// TwinCAT 3 PLC project ReferenceImplementation
// ProgramVersion: 3.1.4026.11
// libraries:
//   Tc2_Standard, * (Beckhoff Automation GmbH)
//   Tc2_System, * (Beckhoff Automation GmbH)
//   Tc3_Module, * (Beckhoff Automation GmbH)
//   [Resi4MPM], * (Jan Wilch)
//   [xPPU], * (Jan Wilch)
// project tree:
//   DUTs/ SRecoveryRequestOutput.TcDUT, STriggeredOutput.TcDUT
//   GVLs/ HMI_Texts.TcGVL, RaInterface_GVL.TcGVL (excluded from build), xPPU_Container.TcPOU
//   / PlcTask.TcTTO
//   POUs/00_ProgramMain/ MAIN.TcPOU
//   POUs/01_SequenceControl/ xPPU_Automatic.TcPOU, xPPU_LSC.TcPOU, xPPU_Crane.TcPOU, xPPU_PAC.TcPOU, xPPU_PicAlpha.TcPOU, xPPU_RFC.TcPOU, xPPU_SSC.TcPOU, xPPU_Stack.TcPOU, xPPU_Stamp.TcPOU
//   POUs/98_Utility/ FC_InitAlarmTexts.TcPOU
//   POUs/99_ExtrafunctionalImpl/ ButtonManager.TcPOU
// real-time tasks:
//   TASK PlcTask: cycle T#10ms, priority 20, ADS port 351
// I/O:
//   DEVICE Device 1 (EtherCAT), AmsNetId 192.168.5.90.2.1
//     Term 84 (EK1200) [EK1200-5000 EtherCAT Power supply (2A E-Bus)]
//       Term 2 (EK1110) [EK1110 EtherCAT extension]
//     BK1 (EK1100) [EK1100 EtherCAT Coupler (2A E-Bus)]
//       1.2 (EL1004) [EL1004 4Ch. Dig. Input 24V, 3ms]
//       1.3 (EL1004) [EL1004 4Ch. Dig. Input 24V, 3ms]
//       1.4 (EL1004) [EL1004 4Ch. Dig. Input 24V, 3ms]
//       1.5 (EL1004) [EL1004 4Ch. Dig. Input 24V, 3ms]
//       1.6 (EL2004) [EL2004 4Ch. Dig. Output 24V, 0.5A]
//       1.9 (EL2004) [EL2004 4Ch. Dig. Output 24V, 0.5A]
//       1.10 (EL2004) [EL2004 4Ch. Dig. Output 24V, 0.5A]
//       1.11 (EL2004) [EL2004 4Ch. Dig. Output 24V, 0.5A]
//       1.12 (EL1004) [EL1004 4Ch. Dig. Input 24V, 3ms]
//       1.13 (EL3162) [EL3162 2Ch. Ana. Input 0-10V]
//       1.14 (EL9011) [EL9011 End Terminal]
//     BK2&3 (EK1100) [EK1100 EtherCAT Coupler (2A E-Bus)]
//       2&3.2 (EL1004) [EL1004 4Ch. Dig. Input 24V, 3ms]
//       2&3.3 (EL1004) [EL1004 4Ch. Dig. Input 24V, 3ms]
//       2&3.4 (EL1004) [EL1004 4Ch. Dig. Input 24V, 3ms]
//       2&3.5 (EL1004) [EL1004 4Ch. Dig. Input 24V, 3ms]
//       2&3.6 (EL1004) [EL1004 4Ch. Dig. Input 24V, 3ms]
//       2&3.7 (EL1004) [EL1004 4Ch. Dig. Input 24V, 3ms]
//       2&3.10 (EL2004) [EL2004 4Ch. Dig. Output 24V, 0.5A]
//       2&3.11 (EL2004) [EL2004 4Ch. Dig. Output 24V, 0.5A]
//       2&3.12 (EL2004) [EL2004 4Ch. Dig. Output 24V, 0.5A]
//       2&3.13 (EL2004) [EL2004 4Ch. Dig. Output 24V, 0.5A]
//       2&3.14 (EL1004) [EL1004 4Ch. Dig. Input 24V, 3ms]
//       2&3.16 (EL4102) [EL4102 2Ch. Ana. Output 0-10V]
//       2&3.17 (EL4102) [EL4102 2Ch. Ana. Output 0-10V]
//       2&3.18 (EL9011) [EL9011 End Terminal]
//     BK4 (EK1100) [EK1100 EtherCAT Coupler (2A E-Bus)]
//       4.2 (EL1808) [EL1808 8Ch. Dig. Input 24V, 3ms]
//       4.3 (EL1004) [EL1004 4Ch. Dig. Input 24V, 3ms]
//       4.4 (EL1004) [EL1004 4Ch. Dig. Input 24V, 3ms]
//       4.5 (EL1004) [EL1004 4Ch. Dig. Input 24V, 3ms]
//       4.6 (EL1004) [EL1004 4Ch. Dig. Input 24V, 3ms]
//       4.7 (EL1004) [EL1004 4Ch. Dig. Input 24V, 3ms]
//       4.8 (EL3064) [EL3064 4Ch. Ana. Input 0-10V]
//       4.9 (EL3064) [EL3064 4Ch. Ana. Input 0-10V]
//       4.10 (EL3164) [EL3164 4Ch. Ana. Input 0-10V]
//       4.11 (EL3054) [EL3054 4Ch. Ana. Input 4-20mA]
//       Term 208 (EL3058) [EL3058 8Ch. Ana. Input 4-20mA]
//       4.13 (EL2004) [EL2004 4Ch. Dig. Output 24V, 0.5A]
//       4.14 (EL2004) [EL2004 4Ch. Dig. Output 24V, 0.5A]
//       4.15 (EL9011) [EL9011 End Terminal]
//     BK5 (EK1100) [EK1100 EtherCAT Coupler (2A E-Bus)]
//       5.2 (EL1008) [EL1008 8Ch. Dig. Input 24V, 3ms]
//       5.3 (EL5152) [EL5152 2Ch. Inc. Encoder]
//       5.6 (EL2008) [EL2008 8Ch. Dig. Output 24V, 0.5A]
//       5.7 (EL4102) [EL4102 2Ch. Ana. Output 0-10V]
//       5.8 (EL9011) [EL9011 End Terminal]
//     BK6 (EK1100) [EK1100 EtherCAT Coupler (2A E-Bus)]
//       6.2 (EL3062) [EL3062 2Ch. Ana. Input 0-10V]
//       6.3 (EL6224) [EL6224 (IO Link Master)]
//       6.4 (EL9011) [EL9011 End Terminal]
//     BK7 (EK1100) [EK1100 EtherCAT Coupler (2A E-Bus)]
//       7.2 (EL1004) [EL1004 4Ch. Dig. Input 24V, 3ms]
//       7.5 (EL2004) [EL2004 4Ch. Dig. Output 24V, 0.5A]
//       7.8 (EL6224) [EL6224 (IO Link Master)]
//       7.9 (EL9011) [EL9011 End Terminal]
//     BK8 (EK1100) [EK1100 EtherCAT Coupler (2A E-Bus)]
//       8.2 (EL1008) [EL1008 8Ch. Dig. Input 24V, 3ms]
//       8.3 (EL1004) [EL1004 4Ch. Dig. Input 24V, 3ms]
//       8.4 (EL3062) [EL3062 2Ch. Ana. Input 0-10V]
//       8.5 (EL2004) [EL2004 4Ch. Dig. Output 24V, 0.5A]
//       8.8 (EL2008) [EL2008 8Ch. Dig. Output 24V, 0.5A]
//       8.9 (EL2004) [EL2004 4Ch. Dig. Output 24V, 0.5A]
//       Term 114 (EL1808) [EL1808 8Ch. Dig. Input 24V, 3ms]
//       8.10 (EL9011) [EL9011 End Terminal]
//     BK9 (EK1100) [EK1100 EtherCAT Coupler (2A E-Bus)]
//       9.2 (EL1004) [EL1004 4Ch. Dig. Input 24V, 3ms]
//       9.3 (EL5152) [EL5152 2Ch. Inc. Encoder]
//       9.6 (EL2004) [EL2004 4Ch. Dig. Output 24V, 0.5A]
//       9.7 (EL4102) [EL4102 2Ch. Ana. Output 0-10V]
//       9.8 (EL9011) [EL9011 End Terminal]
//     BK10 (EK1100) [EK1100 EtherCAT Coupler (2A E-Bus)]
//       10.2 (EL1004) [EL1004 4Ch. Dig. Input 24V, 3ms]
//       10.3 (EL5152) [EL5152 2Ch. Inc. Encoder]
//       10.6 (EL2004) [EL2004 4Ch. Dig. Output 24V, 0.5A]
//       10.7 (EL4102) [EL4102 2Ch. Ana. Output 0-10V]
//       10.8 (EL9011) [EL9011 End Terminal]
//     BK11 (EK1100) [EK1100 EtherCAT Coupler (2A E-Bus)]
//       11.2 (EL1004) [EL1004 4Ch. Dig. Input 24V, 3ms]
//       11.3 (EL3064) [EL3064 4Ch. Ana. Input 0-10V]
//       11.6 (EL2004) [EL2004 4Ch. Dig. Output 24V, 0.5A]
//       11.7 (EL9011) [EL9011 End Terminal]
// variable links:
//   ReferenceImplementation/ReferenceImplementation Instance <-> Device 1 (EtherCAT)/BK1 (EK1100)/1.10 (EL2004)
//     PlcTask Outputs/MAIN.m_container.m_crane.Motor.DO_TurnClockwise <-> Channel 4/Output
//     PlcTask Outputs/MAIN.m_container.m_crane.Motor.DO_TurnCounterclockwise <-> Channel 3/Output
//   ReferenceImplementation/ReferenceImplementation Instance <-> Device 1 (EtherCAT)/BK1 (EK1100)/1.2 (EL1004)
//     PlcTask Inputs/MAIN.m_buttonManager.DI_AutomaticSwitch_StackTerminal <-> Channel 3/Input
//     PlcTask Inputs/MAIN.m_buttonManager.DI_EStopButton_Terminal1 <-> Channel 1/Input
//     PlcTask Inputs/MAIN.m_buttonManager.DI_StartButton_Terminal1 <-> Channel 2/Input
//     PlcTask Inputs/MAIN.m_container.m_crane.o_VacuumGripper.DI_TakenIn <-> Channel 4/Input
//   ReferenceImplementation/ReferenceImplementation Instance <-> Device 1 (EtherCAT)/BK1 (EK1100)/1.3 (EL1004)
//     PlcTask Inputs/MAIN.m_container.m_crane.o_MonostableCylinder.DI_Extended <-> Channel 1/Input
//     PlcTask Inputs/MAIN.m_container.m_crane.o_MonostableCylinder.DI_Retracted <-> Channel 2/Input
//     PlcTask Inputs/MAIN.m_container.m_stack.o_slidingCylinder.DI_Extended <-> Channel 4/Input
//     PlcTask Inputs/MAIN.m_container.m_stack.o_slidingCylinder.DI_Retracted <-> Channel 3/Input
//   ReferenceImplementation/ReferenceImplementation Instance <-> Device 1 (EtherCAT)/BK1 (EK1100)/1.4 (EL1004)
//     PlcTask Inputs/MAIN.m_container.m_crane.m_PresenceSensorAtConveyor.DI_WPDetected <-> Channel 4/Input
//     PlcTask Inputs/MAIN.m_container.m_crane.m_PresenceSensorAtStamp.DI_WPDetected <-> Channel 3/Input
//     PlcTask Inputs/MAIN.m_container.m_stack.m_Inductivesensor.DI_WPMetallic <-> Channel 1/Input
//     PlcTask Inputs/MAIN.m_container.m_stack.m_Opticalsensor.DI_WPLight <-> Channel 2/Input
//   ReferenceImplementation/ReferenceImplementation Instance <-> Device 1 (EtherCAT)/BK1 (EK1100)/1.5 (EL1004)
//     PlcTask Inputs/MAIN.m_container.m_crane.m_PresenceSensorAtStack.DI_WPDetected <-> Channel 1/Input
//     PlcTask Inputs/MAIN.m_container.m_stack.m_Presencesensor.DI_WPDetected <-> Channel 2/Input
//   ReferenceImplementation/ReferenceImplementation Instance <-> Device 1 (EtherCAT)/BK1 (EK1100)/1.6 (EL2004)
//     PlcTask Outputs/MAIN.m_container.m_crane.o_VacuumGripper.DO_VacuumOn <-> Channel 1/Output
//   ReferenceImplementation/ReferenceImplementation Instance <-> Device 1 (EtherCAT)/BK1 (EK1100)/1.9 (EL2004)
//     PlcTask Outputs/MAIN.m_container.m_crane.o_MonostableCylinder.DO_Extend <-> Channel 1/Output
//     PlcTask Outputs/MAIN.m_container.m_stack.o_slidingCylinder.DO_Extend <-> Channel 2/Output
//   ReferenceImplementation/ReferenceImplementation Instance <-> Device 1 (EtherCAT)/BK10 (EK1100)/10.2 (EL1004)
//     PlcTask Inputs/MAIN.m_container.m_SSC.m_PresencesensorEnd.DI_WPDetected <-> Channel 2/Input
//     PlcTask Inputs/MAIN.m_container.m_SSC.m_PresencesensorStart.DI_WPDetected <-> Channel 1/Input
//     PlcTask Inputs/MAIN.m_container.m_SSC.m_Switch.DI_Extended <-> Channel 4/Input
//     PlcTask Inputs/MAIN.m_container.m_SSC.m_Switch.DI_Retracted <-> Channel 3/Input
//   ReferenceImplementation/ReferenceImplementation Instance <-> Device 1 (EtherCAT)/BK10 (EK1100)/10.6 (EL2004)
//     PlcTask Outputs/MAIN.m_container.m_SSC.Motor.DO_TurnClockwise <-> Channel 1/Output
//     PlcTask Outputs/MAIN.m_container.m_SSC.Motor.DO_TurnCounterclockwise <-> Channel 2/Output
//     PlcTask Outputs/MAIN.m_container.m_SSC.m_Switch.DO_Extend <-> Channel 3/Output
//   ReferenceImplementation/ReferenceImplementation Instance <-> Device 1 (EtherCAT)/BK2&3 (EK1100)/2&3.10 (EL2004)
//     PlcTask Outputs/MAIN.m_container.m_stamp.m_slidingCylinder.DO_Extend <-> Channel 1/Output
//     PlcTask Outputs/MAIN.m_container.m_stamp.m_slidingCylinder.DO_Retract <-> Channel 2/Output
//     PlcTask Outputs/MAIN.m_container.m_stamp.m_stampingCylinder.DO_Extend <-> Channel 3/Output
//   ReferenceImplementation/ReferenceImplementation Instance <-> Device 1 (EtherCAT)/BK2&3 (EK1100)/2&3.11 (EL2004)
//     PlcTask Outputs/MAIN.m_container.m_LSC.Motor.DO_TurnClockwise <-> Channel 4/Output
//     PlcTask Outputs/MAIN.m_container.m_LSC.m_rampPusherMid.DO_Extend <-> Channel 3/Output
//     PlcTask Outputs/MAIN.m_container.m_LSC.m_rampPusherStart.DO_Extend <-> Channel 2/Output
//   ReferenceImplementation/ReferenceImplementation Instance <-> Device 1 (EtherCAT)/BK2&3 (EK1100)/2&3.12 (EL2004)
//     PlcTask Outputs/MAIN.m_container.m_LSC.Motor.DO_TurnCounterclockwise <-> Channel 1/Output
//   ReferenceImplementation/ReferenceImplementation Instance <-> Device 1 (EtherCAT)/BK2&3 (EK1100)/2&3.16 (EL4102)
//     PlcTask Outputs/MAIN.m_container.m_stamp.m_pressureValve.AO_SetPressure <-> Channel 2/Output
//   ReferenceImplementation/ReferenceImplementation Instance <-> Device 1 (EtherCAT)/BK2&3 (EK1100)/2&3.2 (EL1004)
//     PlcTask Inputs/MAIN.m_buttonManager.DI_AutomaticSwitch_StampTerminal <-> Channel 1/Input
//     PlcTask Inputs/MAIN.m_container.m_stamp.m_slidingCylinder.DI_Extended <-> Channel 2/Input
//     PlcTask Inputs/MAIN.m_container.m_stamp.m_slidingCylinder.DI_Retracted <-> Channel 3/Input
//     PlcTask Inputs/MAIN.m_container.m_stamp.m_stampingCylinder.DI_Retracted <-> Channel 4/Input
//   ReferenceImplementation/ReferenceImplementation Instance <-> Device 1 (EtherCAT)/BK2&3 (EK1100)/2&3.3 (EL1004)
//     PlcTask Inputs/MAIN.m_buttonManager.DI_EStopButton_Terminal3 <-> Channel 3/Input
//     PlcTask Inputs/MAIN.m_buttonManager.DI_StartButton_Terminal3 <-> Channel 4/Input
//     PlcTask Inputs/MAIN.m_container.m_stamp.m_presenceSensor.DI_WPDetected <-> Channel 2/Input
//     PlcTask Inputs/MAIN.m_container.m_stamp.m_stampingCylinder.DI_Extended <-> Channel 1/Input
//   ReferenceImplementation/ReferenceImplementation Instance <-> Device 1 (EtherCAT)/BK2&3 (EK1100)/2&3.4 (EL1004)
//     PlcTask Inputs/MAIN.m_buttonManager.DI_AutomaticSwitch_LSCTerminal <-> Channel 1/Input
//     PlcTask Inputs/MAIN.m_container.m_LSC.m_inductiveSensorStart.DI_WPMetallic <-> Channel 4/Input
//     PlcTask Inputs/MAIN.m_container.m_LSC.m_presenceSensorStart.DI_WPDetected <-> Channel 3/Input
//   ReferenceImplementation/ReferenceImplementation Instance <-> Device 1 (EtherCAT)/BK2&3 (EK1100)/2&3.5 (EL1004)
//     PlcTask Inputs/MAIN.m_container.m_LSC.m_inductiveSensorMid.DI_WPMetallic <-> Channel 2/Input
//     PlcTask Inputs/MAIN.m_container.m_LSC.m_opticalSensorEnd.DI_WPLight <-> Channel 4/Input
//     PlcTask Inputs/MAIN.m_container.m_LSC.m_opticalSensorMid.DI_WPLight <-> Channel 3/Input
//     PlcTask Inputs/MAIN.m_container.m_LSC.m_opticalSensorStart.DI_WPLight <-> Channel 1/Input
//   ReferenceImplementation/ReferenceImplementation Instance <-> Device 1 (EtherCAT)/BK2&3 (EK1100)/2&3.6 (EL1004)
//     PlcTask Inputs/MAIN.m_container.m_LSC.m_rampPusherMid.DI_Extended <-> Channel 3/Input
//     PlcTask Inputs/MAIN.m_container.m_LSC.m_rampPusherMid.DI_Retracted <-> Channel 4/Input
//     PlcTask Inputs/MAIN.m_container.m_LSC.m_rampPusherStart.DI_Extended <-> Channel 1/Input
//     PlcTask Inputs/MAIN.m_container.m_LSC.m_rampPusherStart.DI_Retracted <-> Channel 2/Input
//   ReferenceImplementation/ReferenceImplementation Instance <-> Device 1 (EtherCAT)/BK2&3 (EK1100)/2&3.7 (EL1004)
//     PlcTask Inputs/MAIN.m_buttonManager.DI_EStopButton_Terminal2 <-> Channel 3/Input
//     PlcTask Inputs/MAIN.m_buttonManager.DI_StartButton_Terminal2 <-> Channel 4/Input
//   ReferenceImplementation/ReferenceImplementation Instance <-> Device 1 (EtherCAT)/BK4 (EK1100)/4.2 (EL1808)
//     PlcTask Inputs/MAIN.m_container.m_LSC.m_rampEnd.m_presenceSensorRampFull.DI_WPDetected <-> Channel 8/Input
//     PlcTask Inputs/MAIN.m_container.m_LSC.m_rampMiddle.m_presenceSensorRampFull.DI_WPDetected <-> Channel 7/Input
//     PlcTask Inputs/MAIN.m_container.m_LSC.m_rampStart.m_presenceSensorRampFull.DI_WPDetected <-> Channel 6/Input
//   ReferenceImplementation/ReferenceImplementation Instance <-> Device 1 (EtherCAT)/BK4 (EK1100)/4.3 (EL1004)
//     PlcTask Inputs/MAIN.m_container.m_stack.o_slidingCylinder.DI_BoundaryPressure <-> Channel 1/Input
//     PlcTask Inputs/MAIN.m_container.m_stamp.m_slidingCylinder.DI_BoundaryPressure <-> Channel 2/Input
//   ReferenceImplementation/ReferenceImplementation Instance <-> Device 1 (EtherCAT)/BK4 (EK1100)/4.4 (EL1004)
//     PlcTask Inputs/MAIN.m_container.m_stamp.m_stampingCylinder.DI_BoundaryPressure <-> Channel 4/Input
//   ReferenceImplementation/ReferenceImplementation Instance <-> Device 1 (EtherCAT)/BK4 (EK1100)/4.5 (EL1004)
//     PlcTask Inputs/MAIN.m_container.m_SSC.m_Inductivesensor.DI_WPMetallic <-> Channel 2/Input
//     PlcTask Inputs/MAIN.m_container.m_SSC.m_Opticalsensor.DI_WPLight <-> Channel 1/Input
//     PlcTask Inputs/MAIN.m_container.m_SSC.m_Ramp.m_presenceSensorRampFull.DI_WPDetected <-> Channel 3/Input
//   ReferenceImplementation/ReferenceImplementation Instance <-> Device 1 (EtherCAT)/BK4 (EK1100)/4.6 (EL1004)
//     PlcTask Inputs/MAIN.m_container.m_stamp.m_stampingCylinder.DI_BoundaryFlowPressure <-> Channel 1/Input
//   ReferenceImplementation/ReferenceImplementation Instance <-> Device 1 (EtherCAT)/BK4 (EK1100)/4.9 (EL3064)
//     PlcTask Inputs/MAIN.m_container.m_stamp.m_pressureSensor.AI_CurrentPressure <-> AI Standard Channel 2/Value
//   ReferenceImplementation/ReferenceImplementation Instance <-> Device 1 (EtherCAT)/BK5 (EK1100)/5.2 (EL1008)
//     PlcTask Inputs/MAIN.m_buttonManager.DI_AutomaticSwitch_DoorTerminal <-> Channel 3/Input
//     PlcTask Inputs/MAIN.m_buttonManager.DI_ResetButton_Door <-> Channel 4/Input
//     PlcTask Inputs/MAIN.m_buttonManager.DI_StartButton_Door <-> Channel 1/Input
//     PlcTask Inputs/MAIN.m_buttonManager.DI_StopButton_Door <-> Channel 2/Input
//     PlcTask Inputs/MAIN.m_container.m_RFC.m_PresencesensorEnd.DI_WPDetected <-> Channel 6/Input
//     PlcTask Inputs/MAIN.m_container.m_RFC.m_PresencesensorStart.DI_WPDetected <-> Channel 5/Input
//     PlcTask Inputs/MAIN.m_container.m_RFC.m_Switch.DI_Extended <-> Channel 8/Input
//     PlcTask Inputs/MAIN.m_container.m_RFC.m_Switch.DI_Retracted <-> Channel 7/Input
//   ReferenceImplementation/ReferenceImplementation Instance <-> Device 1 (EtherCAT)/BK5 (EK1100)/5.6 (EL2008)
//     PlcTask Outputs/MAIN.m_container.m_RFC.Motor.DO_TurnClockwise <-> Channel 5/Output
//     PlcTask Outputs/MAIN.m_container.m_RFC.Motor.DO_TurnCounterclockwise <-> Channel 6/Output
//     PlcTask Outputs/MAIN.m_container.m_RFC.m_Switch.DO_Extend <-> Channel 7/Output
//   ReferenceImplementation/ReferenceImplementation Instance <-> Device 1 (EtherCAT)/BK6 (EK1100)/6.2 (EL3062)
//     PlcTask Inputs/MAIN.m_container.m_stack.m_Weightsensor.AI_WPWeight <-> AI Standard Channel 1/Value
//   ReferenceImplementation/ReferenceImplementation Instance <-> Device 1 (EtherCAT)/BK7 (EK1100)/7.5 (EL2004)
//     PlcTask Outputs/MAIN.m_container.m_LSC.m_Switch.DO_Extend <-> Channel 3/Output
//   ReferenceImplementation/ReferenceImplementation Instance <-> Device 1 (EtherCAT)/BK8 (EK1100)/8.2 (EL1008)
//     PlcTask Inputs/MAIN.m_buttonManager.DI_EStopButton_LightBarrier <-> Channel 8/Input
//     PlcTask Inputs/MAIN.m_container.m_PicAlpha.m_PresenceSensorPosition1.DI_WPDetected <-> Channel 2/Input
//     PlcTask Inputs/MAIN.m_container.m_PicAlpha.m_PresenceSensorPosition2.DI_WPDetected <-> Channel 7/Input
//     PlcTask Inputs/MAIN.m_container.m_PicAlpha.m_PresenceSensorPosition3.DI_WPDetected <-> Channel 4/Input
//     PlcTask Inputs/MAIN.m_container.m_PicAlpha.m_PresenceSensorPosition4.DI_WPDetected <-> Channel 3/Input
//     PlcTask Inputs/MAIN.m_container.m_PicAlpha.o_MonostableCylinder.DI_Extended <-> Channel 5/Input
//     PlcTask Inputs/MAIN.m_container.m_PicAlpha.o_MonostableCylinder.DI_Retracted <-> Channel 6/Input
//     PlcTask Inputs/MAIN.m_container.m_PicAlpha.o_VacuumGripper.DI_TakenIn <-> Channel 1/Input
//   ReferenceImplementation/ReferenceImplementation Instance <-> Device 1 (EtherCAT)/BK8 (EK1100)/8.3 (EL1004)
//     PlcTask Inputs/MAIN.m_buttonManager.DI_AutomaticSwitch_LightGridTerminal <-> Channel 3/Input
//     PlcTask Inputs/MAIN.m_buttonManager.DI_ResetButton_LightBarrier <-> Channel 4/Input
//     PlcTask Inputs/MAIN.m_buttonManager.DI_StartButton_LightBarrier <-> Channel 1/Input
//     PlcTask Inputs/MAIN.m_buttonManager.DI_StopButton_LightBarrier <-> Channel 2/Input
//   ReferenceImplementation/ReferenceImplementation Instance <-> Device 1 (EtherCAT)/BK8 (EK1100)/8.5 (EL2004)
//     PlcTask Outputs/MAIN.m_container.m_PicAlpha.o_VacuumGripper.DO_VacuumOn <-> Channel 1/Output
//   ReferenceImplementation/ReferenceImplementation Instance <-> Device 1 (EtherCAT)/BK8 (EK1100)/8.8 (EL2008)
//     PlcTask Outputs/MAIN.m_container.m_PicAlpha.Motor.DO_TurnClockwise <-> Channel 2/Output
//     PlcTask Outputs/MAIN.m_container.m_PicAlpha.Motor.DO_TurnCounterclockwise <-> Channel 1/Output
//     PlcTask Outputs/MAIN.m_container.m_PicAlpha.o_MonostableCylinder.DO_Extend <-> Channel 3/Output
//     PlcTask Outputs/MAIN.m_container.m_PicAlpha.o_VacuumGripper.VacuumHit <-> Channel 6/Output
//   ReferenceImplementation/ReferenceImplementation Instance <-> Device 1 (EtherCAT)/BK9 (EK1100)/9.2 (EL1004)
//     PlcTask Inputs/MAIN.m_container.m_PAC.m_PresencesensorEnd.DI_WPDetected <-> Channel 2/Input
//     PlcTask Inputs/MAIN.m_container.m_PAC.m_PresencesensorStart.DI_WPDetected <-> Channel 1/Input
//     PlcTask Inputs/MAIN.m_container.m_PAC.m_Switch.DI_Extended <-> Channel 4/Input
//     PlcTask Inputs/MAIN.m_container.m_PAC.m_Switch.DI_Retracted <-> Channel 3/Input
//   ReferenceImplementation/ReferenceImplementation Instance <-> Device 1 (EtherCAT)/BK9 (EK1100)/9.6 (EL2004)
//     PlcTask Outputs/MAIN.m_container.m_PAC.Motor.DO_TurnClockwise <-> Channel 1/Output
//     PlcTask Outputs/MAIN.m_container.m_PAC.Motor.DO_TurnCounterclockwise <-> Channel 2/Output
//     PlcTask Outputs/MAIN.m_container.m_PAC.m_Switch.DO_Extend <-> Channel 3/Output

CONFIGURATION ReferenceImplementation
    RESOURCE PLC ON TwinCAT3
        TASK PlcTask(INTERVAL := T#10ms, PRIORITY := 20);
        PROGRAM MAIN WITH PlcTask : MAIN;
    END_RESOURCE
END_CONFIGURATION

// ---- DUTs/SRecoveryRequestOutput.TcDUT
TYPE SRecoveryRequestOutput EXTENDS STriggeredOutput :
STRUCT
	RequestedState: STRING(256);
END_STRUCT
END_TYPE

// ---- DUTs/STriggeredOutput.TcDUT
TYPE STriggeredOutput :
STRUCT
	ChangeTrigger: USINT;
END_STRUCT
END_TYPE

// ---- GVLs/HMI_Texts.TcGVL
{attribute 'qualified_only'}
VAR_GLOBAL
	AlarmTexts: ARRAY [0..999] OF STRING;
END_VAR

// ---- GVLs/RaInterface_GVL.TcGVL
{attribute 'qualified_only'}
VAR_GLOBAL CONSTANT
	ALARM_ARR_MAX: UINT := 9;
END_VAR

VAR_GLOBAL
	// #################### OUTPUT TO RA ####################
	// alarms detected at field-level or process-level (irregularly pushed to RA)
	{attribute 'OPC.UA.DA' := '1'}
	Out_Alarms: ARRAY [ResiConst.ARR_MIN..RaInterface_GVL.ALARM_ARR_MAX] OF SAlarm;
	
	// the complete set of observed process variables (explicitly checked by RA)
	{attribute 'OPC.UA.DA' := '1'}
	Out_NamedProcessState: ARRAY [ResiConst.ARR_MIN..ResiConst.STATE_ARR_MAX] OF SNamedValue;
	
	// the process state that needs to be restored (irregularly pushed to RA)
	{attribute 'OPC.UA.DA' := '1'}
	{attribute 'OPC.UA.DA.StructuredType' := '1'}
	Out_RecoveryRequest: SRecoveryRequestOutput;
	
	
	// ################### INPUT FROM RA ####################
	// CPA-computed specifications of compensation strategies
	{attribute 'OPC.UA.DA' := '1'}
	In_Compensations: ARRAY [ResiConst.ARR_MIN..ResiConst.COMPENSATIONS_ARR_MAX] OF SCompensation;
	
	// CPA-computed specification of a recovery strategy
	{attribute 'OPC.UA.DA' := '1'}
	{attribute 'OPC.UA.DA.StructuredType' := '1'}
	In_Recovery: SRecovery;
	
	// specifies whether a recovery is ready for execution
	{attribute 'OPC.UA.DA' := '1'}
	In_RecoveryAvailable: BOOL;
	
	// a custom sequence to execute (not the automatic mode)
	{attribute 'OPC.UA.DA' := '1'}
	{attribute 'OPC.UA.DA.StructuredType' := '1'}
	In_CustomSequence: LinearSequence;
	
	// signal the PLC that a custom sequence (not the automatic mode) should be executed
	{attribute 'OPC.UA.DA' := '1'}
	In_RunCustomSequence: BOOL;
	
	// signal the PLC that the custom sequence should be looped infinitely
	{attribute 'OPC.UA.DA' := '1'}
	In_LoopCustomSequence: BOOL;
	
	
	// ################### EDITABLE CONDITIONS ####################
	// Expressions that can be edited by the CPA at runtime
	{attribute 'OPC.UA.DA' := '1'}
	{attribute 'OPC.UA.DA.StructuredType' := '1'}
	In_CompExpressions: ARRAY [ResiConst.ARR_MIN..ResiConst.COMPENSATIONS_ARR_MAX] OF ComparisonExpression(0, EComparisonType.none, EDataType.none, FALSE, 0, '', FALSE);
	{attribute 'OPC.UA.DA' := '1'}
	{attribute 'OPC.UA.DA.StructuredType' := '1'}
	In_ValueExpressions: ARRAY [ResiConst.ARR_MIN..ResiConst.COMPENSATIONS_ARR_MAX] OF ValueExpression(EDataType.none, FALSE, 0, '', FALSE);
	
	// BoolExpressions are described by a "spec" and then actually constructed on the PLC
	// (because otherwise working with the IExpressions left and right is impossible)
	{attribute 'OPC.UA.DA' := '1'}
	{attribute 'OPC.UA.DA.StructuredType' := '1'}
	In_BoolExprSpecs: ARRAY [ResiConst.ARR_MIN..ResiConst.COMPENSATIONS_ARR_MAX] OF SBoolExpressionSpec;
	
	// Specified assignement of specified expressions to primitives (array index = primitive ID)
	// (must be actually assigned on the PLC) 
	{attribute 'OPC.UA.DA' := '1'}
	{attribute 'OPC.UA.DA.StructuredType' := '1'}
	In_RuntimeConditions: ARRAY [ResiConst.ARR_MIN..ResiConst.COMPENSATIONS_ARR_MAX] OF SRuntimeCondition;
END_VAR

// ---- POUs/00_ProgramMain/MAIN.TcPOU
PROGRAM MAIN
VAR CONSTANT
	INSTANCE_NAME: STRING := 'MAIN Program';
	IGNORE_DEFINITION: BOOL := TRUE;
	IGNORE_STOP: BOOL := TRUE;
END_VAR
VAR
	// define services
	m_buttonManager: ButtonManager;
	m_errorManager: ErrorManager;
	m_services: ServiceContainer(ADR(m_errorManager));
	
	// instantiate machine behavior model
	m_container: xPPU_Container(
		m_services.PtrStateTracker, 
		m_services.PtrProcessManager, 
		ADR(m_errorManager));
	
	// INTERLOCKS - must always be False
	// (EProcessVariables.LSC_RampEndWPCount >= 3) AND ((EProcessVariables.LSC_RampStartWPCount >= 3) OR ((EProcessVariables.LSC_RampMiddleWPCount >= 3) OR (EProcessVariables.SSC_RampWPCount >= 3)))
	m_compExpr1: ComparisonExpression(EProcessVariables.LSC_RampEndWPCount, EComparisonType.greater_eq, EDataType.numeric, FALSE, 3, '', TRUE);
	m_compExpr3: ComparisonExpression(EProcessVariables.LSC_RampStartWPCount, EComparisonType.greater_eq, EDataType.numeric, FALSE, 3, '', TRUE);
	m_compExpr5: ComparisonExpression(EProcessVariables.LSC_RampMiddleWPCount, EComparisonType.greater_eq, EDataType.numeric, FALSE, 3, '', TRUE);
	m_compExpr7: ComparisonExpression(EProcessVariables.SSC_RampWPCount, EComparisonType.greater_eq, EDataType.numeric, FALSE, 3, '', TRUE);
	m_boolExpr8: BoolExpression(m_compExpr5, EBoolOperation.or_op, m_compExpr7);
	m_boolExpr9: BoolExpression(m_compExpr3, EBoolOperation.or_op, m_boolExpr8);
	m_allRampsFull: BoolExpression(m_compExpr1, EBoolOperation.and_op, m_boolExpr9);
	
	// INTERLOCKS - must always be True
	// ...
	
	// MANUAL STRATEGY
	m_startAuto: BOOL;
	m_startManual: BOOL;
	m_stopManual: BOOL;
	m_strategyState: EOperationResult;
	
	// other
	i: UINT;
	m_statesEnum: EProcessVariables;
	m_emptyParams: ParameterSet;
	m_didFinishPrimitives: BOOL;
	m_appInitialized: BOOL;
	m_xPPU: xPPU_Automatic;
	m_customSeqStatus: EOperationResult;
	m_steps: ARRAY [0..2] OF STRING;
	m_appObservation: ARRAY[EProcessVariables.operating_mode..EProcessVariables.operating_mode] OF SValue;
END_VAR

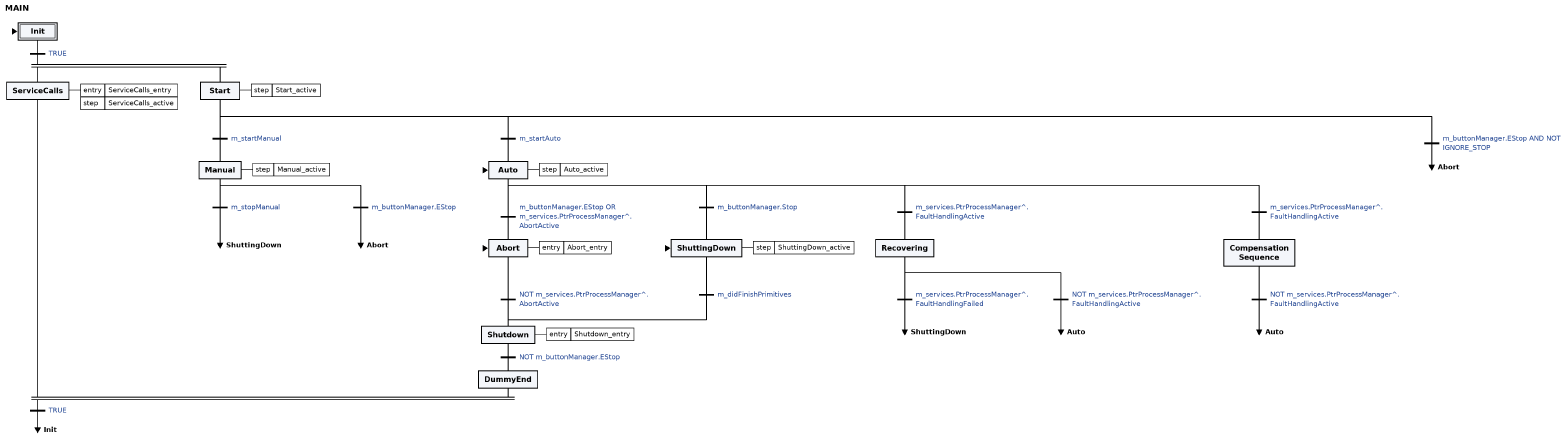
INITIAL_STEP Init:
END_STEP
TRANSITION FROM Init TO (ServiceCalls, Start)
    := TRUE;
END_TRANSITION
STEP ServiceCalls:
    ServiceCalls_entry(P1);  // entry action
    ServiceCalls_active(N);  // step action
END_STEP
STEP Start:
    Start_active(N);  // step action
END_STEP
TRANSITION FROM Start TO Manual
    := m_startManual;
END_TRANSITION
STEP Manual:
    Manual_active(N);  // step action
END_STEP
TRANSITION FROM Manual TO ShuttingDown
    := m_stopManual;
END_TRANSITION
TRANSITION FROM Manual TO Abort
    := m_buttonManager.EStop;
END_TRANSITION
TRANSITION FROM Start TO Auto
    := m_startAuto;
END_TRANSITION
STEP Auto:
    Auto_active(N);  // step action
END_STEP
TRANSITION FROM Auto TO Abort
    := m_buttonManager.EStop OR m_services.PtrProcessManager^.AbortActive;
END_TRANSITION
STEP Abort:
    Abort_entry(P1);  // entry action
END_STEP
TRANSITION FROM Abort TO Shutdown
    := NOT m_services.PtrProcessManager^.AbortActive;
END_TRANSITION
TRANSITION FROM Auto TO ShuttingDown
    := m_buttonManager.Stop;
END_TRANSITION
STEP ShuttingDown:
    ShuttingDown_active(N);  // step action
END_STEP
TRANSITION FROM ShuttingDown TO Shutdown
    := m_didFinishPrimitives;
END_TRANSITION
TRANSITION FROM Auto TO Recovering
    := m_services.PtrProcessManager^.FaultHandlingActive;
END_TRANSITION
STEP Recovering:
END_STEP
TRANSITION FROM Recovering TO ShuttingDown
    := m_services.PtrProcessManager^.FaultHandlingFailed;
END_TRANSITION
TRANSITION FROM Recovering TO Auto
    := NOT m_services.PtrProcessManager^.FaultHandlingActive;
END_TRANSITION
TRANSITION FROM Auto TO CompensationSequence
    := m_services.PtrProcessManager^.FaultHandlingActive;
END_TRANSITION
STEP CompensationSequence:
END_STEP
TRANSITION FROM CompensationSequence TO Auto
    := NOT m_services.PtrProcessManager^.FaultHandlingActive;
END_TRANSITION
STEP Shutdown:
    Shutdown_entry(P1);  // entry action
END_STEP
TRANSITION FROM Shutdown TO DummyEnd
    := NOT m_buttonManager.EStop;
END_TRANSITION
TRANSITION FROM Start TO Abort
    := m_buttonManager.EStop AND NOT IGNORE_STOP;
END_TRANSITION
STEP DummyEnd:
END_STEP
TRANSITION FROM (ServiceCalls, DummyEnd) TO Init
    := TRUE;
END_TRANSITION

ACTION Abort_entry:
m_services.PtrProcessManager^.RequestAbort();
END_ACTION

ACTION Auto_active:
m_xPPU(
	i_ptrErrorManager := m_services.PtrErrorManager,
	i_ptrProcessManager := m_services.PtrProcessManager,
	i_ptrStateTracker := m_services.PtrStateTracker);
END_ACTION

ACTION Manual_active:


m_strategyState := m_services.PtrProcessManager^.ExecuteCustomStrategy();
m_stopManual := m_buttonManager.Stop 
	OR NOT m_services.PtrProcessManager^.CustomStrategyReady 
	OR m_strategyState = EOperationResult.success;
END_ACTION

ACTION ServiceCalls_active:
// process state observation
m_appObservation[EProcessVariables.operating_mode].DataType := EDataType.string_t;
m_appObservation[EProcessVariables.operating_mode].Value.String_t := SFCCurrentStep;

// cylic service updates
IF m_services.PtrStateTracker <>0 THEN
m_services.PtrStateTracker^.CyclicUpdateStatus(IGNORE_DEFINITION,m_appObservation);
m_services.PtrProcessManager^.CyclicManageBehavior();
END_IF
END_ACTION

ACTION ServiceCalls_entry:
IF NOT m_appInitialized THEN
	FC_InitAlarmTexts();
	
	// init process variable names
	FOR i := ResiConst.ARR_MIN TO ResiConst.STATE_ARR_MAX DO
		m_statesEnum := i;
		m_services.PtrStateTracker^.SetProcessVariableName(i, TO_STRING(m_statesEnum));
	END_FOR
	
	// add interlocks
	m_services.PtrStateTracker^.AddInterlock(m_allRampsFull, FALSE);
	
	m_appInitialized := TRUE;
	m_errorManager.AddMessage(EAlarms.initialized, TRUE, ESeverity.info, 'MAIN');
END_IF
END_ACTION

ACTION Shutdown_entry:
m_errorManager.AddMessage(
	i_alarmId := EAlarms.stopped,
	i_active := TRUE,
	i_severity := ESeverity.info,
	i_instanceName := INSTANCE_NAME);

m_services.PtrStateTracker^.ResetDefinitions();
END_ACTION

ACTION ShuttingDown_active:
m_didFinishPrimitives := m_services.PtrProcessManager^.FinishPrimitives(i_abortRecoveries := TRUE);
END_ACTION

ACTION Start_active:
m_startManual := m_buttonManager.Mode = EOperatingModes.manual AND m_services.PtrProcessManager^.CustomStrategyReady AND m_buttonManager.Start;
m_startAuto := m_buttonManager.Mode = EOperatingModes.automatic AND m_buttonManager.Start;
END_ACTION

END_PROGRAM

// ---- POUs/99_ExtrafunctionalImpl/ButtonManager.TcPOU
FUNCTION_BLOCK ButtonManager
VAR_INPUT
END_VAR
VAR_OUTPUT
END_VAR
VAR
	DI_StartButton_Terminal1 AT%I*: BOOL;
	DI_StartButton_Terminal2 AT%I*: BOOL;	
	DI_StartButton_Terminal3 AT%I*: BOOL;	
	DI_StartButton_Door AT%I*: BOOL;	
	DI_StartButton_LightBarrier AT%I*: BOOL;	
	
	DI_StopButton_Door AT%I*: BOOL;	
	DI_StopButton_LightBarrier AT%I*: BOOL;	
	
	DI_AutomaticSwitch_StackTerminal AT%I*: BOOL;
	DI_AutomaticSwitch_StampTerminal AT%I*: BOOL;
	DI_AutomaticSwitch_LSCTerminal AT%I*: BOOL;
	DI_AutomaticSwitch_DoorTerminal AT%I*: BOOL;
	DI_AutomaticSwitch_LightGridTerminal AT%I*: BOOL;
	
	DI_EStopButton_Terminal1 AT%I*: BOOL;
	DI_EStopButton_Terminal2 AT%I*: BOOL;	
	DI_EStopButton_Terminal3 AT%I*: BOOL;	
	//DI_EStopButton_Door AT%I*: BOOL;     //currently not connected to PLC
	DI_EStopButton_LightBarrier AT%I*: BOOL;
	
	DI_ResetButton_Door AT%I*: BOOL;
	DI_ResetButton_LightBarrier AT%I*: BOOL;
END_VAR

//manages the Start-, Stop-, Reset- and EStop-Buttons

PROPERTY EStop : BOOL
GET
// EStops physically implemented as Failsafe, they return True, when not pressed.
//for better handling this is reversed here
EStop := NOT DI_EStopButton_LightBarrier OR NOT DI_EStopButton_Terminal1 OR NOT DI_EStopButton_Terminal2 OR NOT DI_EStopButton_Terminal3;
END_GET
END_PROPERTY

PROPERTY Mode : EOperatingModes
GET
IF DI_AutomaticSwitch_StackTerminal AND DI_AutomaticSwitch_StampTerminal AND DI_AutomaticSwitch_LSCTerminal AND DI_AutomaticSwitch_DoorTerminal AND DI_AutomaticSwitch_LightGridTerminal THEN
	Mode := EOperatingModes.automatic;
ELSIF NOT (DI_AutomaticSwitch_StackTerminal OR DI_AutomaticSwitch_StampTerminal OR DI_AutomaticSwitch_LSCTerminal OR DI_AutomaticSwitch_DoorTerminal OR DI_AutomaticSwitch_LightGridTerminal) THEN
	Mode := EOperatingModes.manual;
ELSE
	Mode := EOperatingModes.none;
END_IF
END_GET
END_PROPERTY

PROPERTY Reset : BOOL
GET
Reset := DI_ResetButton_Door OR DI_ResetButton_LightBarrier;
END_GET
END_PROPERTY

PROPERTY Start : BOOL
GET
Start := DI_StartButton_Door OR DI_StartButton_LightBarrier OR DI_StartButton_Terminal1 OR DI_StartButton_Terminal2 OR DI_StartButton_Terminal3;
END_GET
END_PROPERTY

PROPERTY Stop : BOOL
GET
// EStops physically implemented as Failsafe, they return True, when not pressed.
//for better handling this is reversed here
Stop := NOT DI_StopButton_Door OR NOT DI_StopButton_LightBarrier;
END_GET
END_PROPERTY

END_FUNCTION_BLOCK

// ---- GVLs/xPPU_Container.TcPOU
FUNCTION_BLOCK xPPU_Container
VAR_INPUT
END_VAR
VAR_OUTPUT
END_VAR
VAR
	// hardware control POUs
	m_crane: Crane;
	m_stack: Stack;
	m_stamp: Stamp;
	m_LSC: LargeSortingConveyor;
	m_PAC: PicAlphaConveyor;
	m_PicAlpha: PicAlpha;
	m_SSC: SmallSortingConveyor;
	m_RFC: RefeedingConveyor;
	
	// products
	(*m_craneWP: xPPUProduct;
	m_stackWP: xPPUProduct;
	m_stampWP: xPPUProduct;
	m_LSCWP: xPPUProduct;
	m_PACWP1: xPPUProduct;
	m_PACWP2: xPPUProduct;
	m_PACWP3: xPPUProduct;
	m_PicAlphaWP: xPPUProduct;
	m_SSCWP1: xPPUProduct;
	m_SSCWP2: xPPUProduct;
	m_RFCWP1: xPPUProduct;
	m_RFCWP2: xPPUProduct;*)
	
	m_iCraneWP: xPPUProduct(EProcessVariables.Crane_ProductType);
	m_iStackWP: xPPUProduct(EProcessVariables.Stack_ProductType) ;
	m_iStampWP: xPPUProduct(EProcessVariables.Stamp_ProductType);
	m_iLSCWP: xPPUProduct(EProcessVariables.LSC_ProductType);
	m_iPACWP1: xPPUProduct(EProcessVariables.PAC_ProductType_1);
	m_iPACWP2: xPPUProduct(EProcessVariables.PAC_ProductType_2);
	m_iPACWP3: xPPUProduct(EProcessVariables.PAC_ProductType_3);	
	m_iPicAlphaWP: xPPUProduct(EProcessVariables.PAC_ProductType_1);
	m_iSSCWP1: xPPUProduct(EProcessVariables.SSC_ProductType_1);
	m_iSSCWP2: xPPUProduct(EProcessVariables.SSC_ProductType_2);
	m_iRFCWP1: xPPUProduct(EProcessVariables.RFC_ProductType_1) ;
	m_iRFCWP2: xPPUProduct(EProcessVariables.RFC_ProductType_2);
	
	// hardware observation (if not included in hardware control)
	m_observeCrane: ObserveCrane(ADR(m_crane), ADR(m_iCraneWP));
	m_observeStack: ObserveStack(ADR(m_stack), ADR(m_iStackWP));
	m_observeStamp: ObserveStamp(ADR(m_stamp), ADR(m_iStampWP));
	m_observeLSC: ObserveLSC(ADR(m_LSC), ADR(m_iLSCWP));
	m_observePAC: ObservePAC(ADR(m_PAC), ADR(m_iPACWP1), ADR(m_iPACWP2), ADR(m_iPACWP3));
	m_observePicAlpha: ObservePicAlpha(ADR(m_PicAlpha), ADR(m_iPicAlphaWP));
	m_observeSSC: ObserveSSC(ADR(m_SSC), ADR(m_iSSCWP1), ADR(m_iSSCWP2));
	m_observeRFC: ObserveRFC(ADR(m_RFC), ADR(m_iRFCWP1), ADR(m_iRFCWP2));
	
	// control primitives
	m_craneMoveToStack: Crane_MoveToStack(ADR(m_crane));
	m_craneMoveToStamp: Crane_MoveToStamp(ADR(m_crane));
	m_craneMoveToLSC: Crane_MoveToLSC(ADR(m_crane));
	m_cranePickUpWP: Crane_PickUpWP(ADR(m_crane));
	m_cranePutDownWP: Crane_PutDownWP(ADR(m_crane));
	
	m_stackProvide: Stack_ProvideWorkpiece(ADR(m_stack));
	
	m_stampStamp: Stamp_StampWorkpiece(ADR(m_stamp));
	
	m_LSCTransferWPToRampStart: LSC_TransferWorkpieceTo_RampStart(ADR(m_LSC));
	m_LSCTransferWPToRampMid: LSC_TransferWorkpieceTo_RampMid(ADR(m_LSC));
	m_LSCTransferWPToRampEnd: LSC_TransferWorkpieceTo_RampEnd(ADR(m_LSC));
	m_LSCTransferWPToPAC: LSC_TransferWorkpieceTo_PAC(ADR(m_LSC));
	m_LSCSearchWorkpiece: LSC_SearchWorkpiece(ADR(m_LSC));
	
	m_PACTransferWPToSSC: PAC_TransferWorkpieceTo_SSC(ADR(m_PAC));
	m_PACTransferWPToPSStart: PAC_TransferWorkpieceTo_PSStart(ADR(m_PAC));
	m_PACTransferWPToPSEnd: PAC_TransferWorkpieceTo_PSEnd(ADR(m_PAC));
	
	m_picAlphaMoveToPos1: PicAlpha_MoveToPos1(ADR(m_picAlpha));
	m_picAlphaMoveToPos2: PicAlpha_MoveToPos2(ADR(m_picAlpha));
	m_picAlphaMoveToPos3: PicAlpha_MoveToPos3(ADR(m_picAlpha));
	m_picAlphaMoveToPos4: PicAlpha_MoveToPos4(ADR(m_picAlpha));
	m_picAlphaPickUpWP: PicAlpha_PickUpWP(ADR(m_picAlpha));
	m_picAlphaPutDownWP: PicAlpha_PutDownWP(ADR(m_picAlpha), ADR(m_PAC));
	
	m_SSCTransferWPToPSStart: SSC_TransferWorkpieceTo_PSStart(ADR(m_SSC));
	m_SSCTransferWPToRampEnd: SSC_TransferWorkpieceTo_RampEnd(ADR(m_SSC));
	m_SSCTransferWPToRFC: SSC_TransferWorkpieceTo_RFC(ADR(m_SSC));
	
	m_RFCTransferWPToLSC: RFC_TransferWorkpieceTo_LSC(ADR(m_RFC));
	m_RFCTransferWPToPSEnd: RFC_TransferWorkpieceTo_PSEnd(ADR(m_RFC));
	
	// module sequences
END_VAR

METHOD FB_init : BOOL
VAR_INPUT
	bInitRetains : BOOL; // if TRUE, the retain variables are initialized (warm start / cold start)
	bInCopyCode : BOOL;  // if TRUE, the instance afterwards gets moved into the copy code (online change)

	i_ptrStateTracker: POINTER TO StateTracker;
	i_ptrProcessManager: POINTER TO ProcessManager;
	
	i_ptrErrorManager: POINTER TO ErrorManager;
END_VAR
// provide Services to Behaviors
m_craneMoveToStack.ProvideServices(i_ptrProcessManager,i_ptrStateTracker);
m_craneMoveToStamp.ProvideServices(i_ptrProcessManager,i_ptrStateTracker);
m_craneMoveToLSC.ProvideServices(i_ptrProcessManager,i_ptrStateTracker);
m_cranePickUpWP.ProvideServices(i_ptrProcessManager,i_ptrStateTracker);
m_cranePutDownWP.ProvideServices(i_ptrProcessManager,i_ptrStateTracker);

m_stackProvide.ProvideServices(i_ptrProcessManager,i_ptrStateTracker);

m_stampStamp.ProvideServices(i_ptrProcessManager, i_ptrStateTracker);

m_LSCTransferWPToRampStart.ProvideServices(i_ptrProcessManager, i_ptrStateTracker);
m_LSCTransferWPToRampMid.ProvideServices(i_ptrProcessManager, i_ptrStateTracker);
m_LSCTransferWPToRampEnd.ProvideServices(i_ptrProcessManager, i_ptrStateTracker);
m_LSCTransferWPToPAC.ProvideServices(i_ptrProcessManager, i_ptrStateTracker);
m_LSCSearchWorkpiece.ProvideServices(i_ptrProcessManager, i_ptrStateTracker);

m_PACTransferWPToSSC.ProvideServices(i_ptrProcessManager, i_ptrStateTracker);
m_PACTransferWPToPSStart.ProvideServices(i_ptrProcessManager, i_ptrStateTracker);
m_PACTransferWPToPSEnd.ProvideServices(i_ptrProcessManager, i_ptrStateTracker);

m_picAlphaMoveToPos1.ProvideServices(i_ptrProcessManager, i_ptrStateTracker);
m_picAlphaMoveToPos2.ProvideServices(i_ptrProcessManager, i_ptrStateTracker);
m_picAlphaMoveToPos3.ProvideServices(i_ptrProcessManager, i_ptrStateTracker);
m_picAlphaMoveToPos4.ProvideServices(i_ptrProcessManager, i_ptrStateTracker);
m_picAlphaPickUpWP.ProvideServices(i_ptrProcessManager, i_ptrStateTracker);
m_picAlphaPutDownWP.ProvideServices(i_ptrProcessManager, i_ptrStateTracker);

m_SSCTransferWPToPSStart.ProvideServices(i_ptrProcessManager, i_ptrStateTracker);
m_SSCTransferWPToRampEnd.ProvideServices(i_ptrProcessManager, i_ptrStateTracker);
m_SSCTransferWPToRFC.ProvideServices(i_ptrProcessManager, i_ptrStateTracker);

m_RFCTransferWPToPSEnd.ProvideServices(i_ptrProcessManager, i_ptrStateTracker);
m_RFCTransferWPToLSC.ProvideServices(i_ptrProcessManager, i_ptrStateTracker);

// provide Behaviors to the Process Manager
i_ptrProcessManager^.AddPrimitive(ADR(m_craneMoveToStack));
i_ptrProcessManager^.AddPrimitive(ADR(m_craneMoveToStamp));
i_ptrProcessManager^.AddPrimitive(ADR(m_craneMoveToLSC));
i_ptrProcessManager^.AddPrimitive(ADR(m_cranePickUpWP));
i_ptrProcessManager^.AddPrimitive(ADR(m_cranePutDownWP));

i_ptrProcessManager^.AddPrimitive(ADR(m_stackProvide));

i_ptrProcessManager^.AddPrimitive(ADR(m_stampStamp));

i_ptrProcessManager^.AddPrimitive(ADR(m_LSCTransferWPToRampStart));
i_ptrProcessManager^.AddPrimitive(ADR(m_LSCTransferWPToRampMid));
i_ptrProcessManager^.AddPrimitive(ADR(m_LSCTransferWPToRampEnd));
i_ptrProcessManager^.AddPrimitive(ADR(m_LSCTransferWPToPAC));
i_ptrProcessManager^.AddPrimitive(ADR(m_LSCSearchWorkpiece));

i_ptrProcessManager^.AddPrimitive(ADR(m_PACTransferWPToPSStart));
i_ptrProcessManager^.AddPrimitive(ADR(m_PACTransferWPToPSEnd));
i_ptrProcessManager^.AddPrimitive(ADR(m_PACTransferWPToSSC));

i_ptrProcessManager^.AddPrimitive(ADR(m_picAlphaMoveToPos1));
i_ptrProcessManager^.AddPrimitive(ADR(m_picAlphaMoveToPos2));
i_ptrProcessManager^.AddPrimitive(ADR(m_picAlphaMoveToPos3));
i_ptrProcessManager^.AddPrimitive(ADR(m_picAlphaMoveToPos4));
i_ptrProcessManager^.AddPrimitive(ADR(m_picAlphaPickUpWP));
i_ptrProcessManager^.AddPrimitive(ADR(m_picAlphaPutDownWP));

i_ptrProcessManager^.AddPrimitive(ADR(m_SSCTransferWPToPSStart));
i_ptrProcessManager^.AddPrimitive(ADR(m_SSCTransferWPToRampEnd));
i_ptrProcessManager^.AddPrimitive(ADR(m_SSCTransferWPToRFC));

i_ptrProcessManager^.AddPrimitive(ADR(m_RFCTransferWPToPSEnd));
i_ptrProcessManager^.AddPrimitive(ADR(m_RFCTransferWPToLSC));

// provide observations to the Process Manager
i_ptrStateTracker^.AddObservation(ADR(m_observeCrane));
i_ptrStateTracker^.AddObservation(ADR(m_observeStack));
i_ptrStateTracker^.AddObservation(ADR(m_observeStamp));
i_ptrStateTracker^.AddObservation(ADR(m_observeLSC));
i_ptrStateTracker^.AddObservation(ADR(m_observePAC));
i_ptrStateTracker^.AddObservation(ADR(m_observePicAlpha));
i_ptrStateTracker^.AddObservation(ADR(m_observeSSC));
i_ptrStateTracker^.AddObservation(ADR(m_observeRFC));

// provide workpieces to the Process Manager
i_ptrStateTracker^.RegisterLocalProduct(EProducts.crane_product, ADR(m_iCraneWP));
i_ptrStateTracker^.RegisterLocalProduct(EProducts.stack_product, ADR(m_iStackWP));
i_ptrStateTracker^.RegisterLocalProduct(EProducts.stamp_product, ADR(m_iStampWP));
i_ptrStateTracker^.RegisterLocalProduct(EProducts.LSC_product, ADR(m_iLSCWP));
i_ptrStateTracker^.RegisterLocalProduct(EProducts.PAC_product1, ADR(m_iPACWP1));
i_ptrStateTracker^.RegisterLocalProduct(EProducts.PAC_product2, ADR(m_iPACWP2));
i_ptrStateTracker^.RegisterLocalProduct(EProducts.PAC_product3, ADR(m_iPACWP3));
i_ptrStateTracker^.RegisterLocalProduct(EProducts.PicAlpha_product, ADR(m_iPicAlphaWP));
i_ptrStateTracker^.RegisterLocalProduct(EProducts.RFC_product1, ADR(m_iRFCWP1));
i_ptrStateTracker^.RegisterLocalProduct(EProducts.RFC_product2, ADR(m_iRFCWP2));
i_ptrStateTracker^.RegisterLocalProduct(EProducts.SSC_product1, ADR(m_iSSCWP1));
i_ptrStateTracker^.RegisterLocalProduct(EProducts.SSC_product2, ADR(m_iSSCWP2));
END_METHOD

END_FUNCTION_BLOCK

// ---- POUs/01_SequenceControl/xPPU_Automatic.TcPOU
FUNCTION_BLOCK xPPU_Automatic
VAR CONSTANT
	m_instanceName: STRING := 'xPPU Stamp Workpieces';
END_VAR
VAR_INPUT
	i_ptrErrorManager: POINTER TO ErrorManager;
	i_ptrProcessManager: POINTER TO ProcessManager;
	i_ptrStateTracker: POINTER TO StateTracker;
END_VAR
VAR
	m_stack: xPPU_Stack;
	m_crane: xPPU_Crane;
	m_stamp: xPPU_Stamp;
	m_LSC: xPPU_LSC;
	m_PAC: xPPU_PAC;
	m_PicAlpha: xPPU_PicAlpha;
	m_SSC: xPPU_SSC;
	m_RFC: xPPU_RFC;
END_VAR

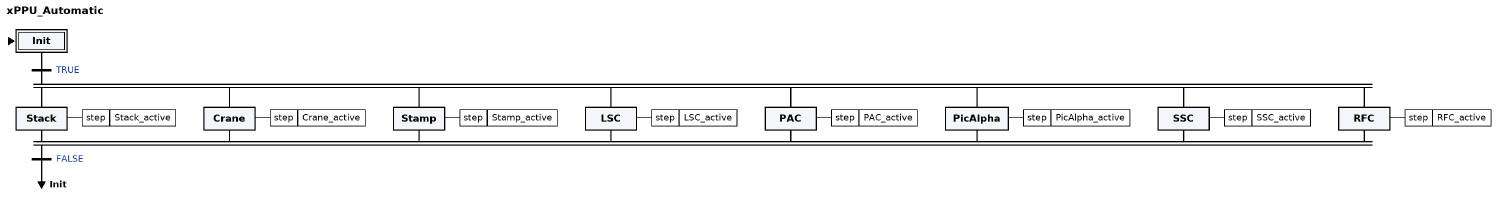
INITIAL_STEP Init:
END_STEP
TRANSITION FROM Init TO (Stack, Crane, Stamp, LSC, PAC, PicAlpha, SSC, RFC)
    := TRUE;
END_TRANSITION
STEP Stack:
    Stack_active(N);  // step action
END_STEP
STEP Crane:
    Crane_active(N);  // step action
END_STEP
STEP Stamp:
    Stamp_active(N);  // step action
END_STEP
STEP LSC:
    LSC_active(N);  // step action
END_STEP
STEP PAC:
    PAC_active(N);  // step action
END_STEP
STEP PicAlpha:
    PicAlpha_active(N);  // step action
END_STEP
STEP SSC:
    SSC_active(N);  // step action
END_STEP
STEP RFC:
    RFC_active(N);  // step action
END_STEP
TRANSITION FROM (Stack, Crane, Stamp, LSC, PAC, PicAlpha, SSC, RFC) TO Init
    := FALSE;
END_TRANSITION

ACTION Crane_active:
m_crane(
	i_error := i_ptrErrorManager, 
	i_process := i_ptrProcessManager,
	i_state := i_ptrStateTracker);
END_ACTION

ACTION LSC_active:
m_LSC(
	i_error := i_ptrErrorManager, 
	i_process := i_ptrProcessManager,
	i_state := i_ptrStateTracker);
END_ACTION

ACTION PAC_active:
m_PAC(
	i_error := i_ptrErrorManager, 
	i_process := i_ptrProcessManager,
	i_state := i_ptrStateTracker);
END_ACTION

ACTION PicAlpha_active:
m_PicAlpha(
	i_error := i_ptrErrorManager, 
	i_process := i_ptrProcessManager,
	i_state := i_ptrStateTracker);
END_ACTION

ACTION RFC_active:
// TODO - this messes up the screwdriver demo! (deactivated for now)

//m_RFC(
//	i_error := i_ptrErrorManager, 
//	i_process := i_ptrProcessManager,
//	i_state := i_ptrStateTracker);
END_ACTION

ACTION SSC_active:
m_SSC(
	i_error := i_ptrErrorManager, 
	i_process := i_ptrProcessManager,
	i_state := i_ptrStateTracker);
END_ACTION

ACTION Stack_active:
m_stack(
	i_error := i_ptrErrorManager, 
	i_process := i_ptrProcessManager,
	i_state := i_ptrStateTracker);
END_ACTION

ACTION Stamp_active:
m_stamp(
	i_error := i_ptrErrorManager, 
	i_process := i_ptrProcessManager,
	i_state := i_ptrStateTracker);
END_ACTION

PROPERTY SubSteps : ARRAY [0..2] OF STRING
GET
VAR
	m_tmp: ARRAY [0..2] OF STRING;
END_VAR
m_tmp[0] := TO_STRING(m_stack.SFCCurrentStep);
m_tmp[1] := TO_STRING(m_crane.SFCCurrentStep);
m_tmp[2] := TO_STRING(m_stamp.SFCCurrentStep);
SubSteps := m_tmp;
END_GET
END_PROPERTY

END_FUNCTION_BLOCK

// ---- POUs/01_SequenceControl/xPPU_Stack.TcPOU
FUNCTION_BLOCK xPPU_Stack
VAR CONSTANT
	IGNORE_EMPTY: BOOL := TRUE;
END_VAR
VAR_INPUT
	i_error: POINTER TO ErrorManager;
	i_process: POINTER TO ProcessManager;
	i_state: POINTER TO StateTracker;
END_VAR
VAR
	m_emptyParams: ParameterSet;
	m_subRes: EOperationResult;
END_VAR

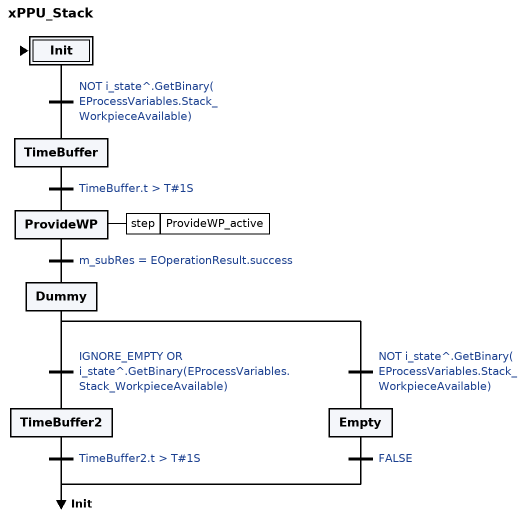
INITIAL_STEP Init:
END_STEP
TRANSITION FROM Init TO TimeBuffer
    := NOT i_state^.GetBinary(EProcessVariables.Stack_WorkpieceAvailable);
END_TRANSITION
STEP TimeBuffer:
END_STEP
TRANSITION FROM TimeBuffer TO ProvideWP
    := TimeBuffer.t > T#1S;
END_TRANSITION
STEP ProvideWP:
    ProvideWP_active(N);  // step action
END_STEP
TRANSITION FROM ProvideWP TO Dummy
    := m_subRes = EOperationResult.success;
END_TRANSITION
STEP Dummy:
END_STEP
TRANSITION FROM Dummy TO TimeBuffer2
    := IGNORE_EMPTY OR i_state^.GetBinary(EProcessVariables.Stack_WorkpieceAvailable);
END_TRANSITION
STEP TimeBuffer2:
END_STEP
TRANSITION FROM TimeBuffer2 TO Init
    := TimeBuffer2.t > T#1S;
END_TRANSITION
TRANSITION FROM Dummy TO Empty
    := NOT i_state^.GetBinary(EProcessVariables.Stack_WorkpieceAvailable);
END_TRANSITION
STEP Empty:
END_STEP
TRANSITION FROM Empty TO Init
    := FALSE;
END_TRANSITION

ACTION ProvideWP_active:
m_subRes := i_process^.Execute(
	EBehaviorType.control_primitive,
	EPrimitives.Stack_ProvideWorkpiece,
	m_emptyParams);
END_ACTION

END_FUNCTION_BLOCK

// ---- POUs/01_SequenceControl/xPPU_Crane.TcPOU
FUNCTION_BLOCK xPPU_Crane
VAR_INPUT
	i_error: POINTER TO ErrorManager;
	i_process: POINTER TO ProcessManager;
	i_state: POINTER TO StateTracker;
END_VAR
VAR
	m_emptyParams: ParameterSet;
	m_subRes: EOperationResult;
END_VAR

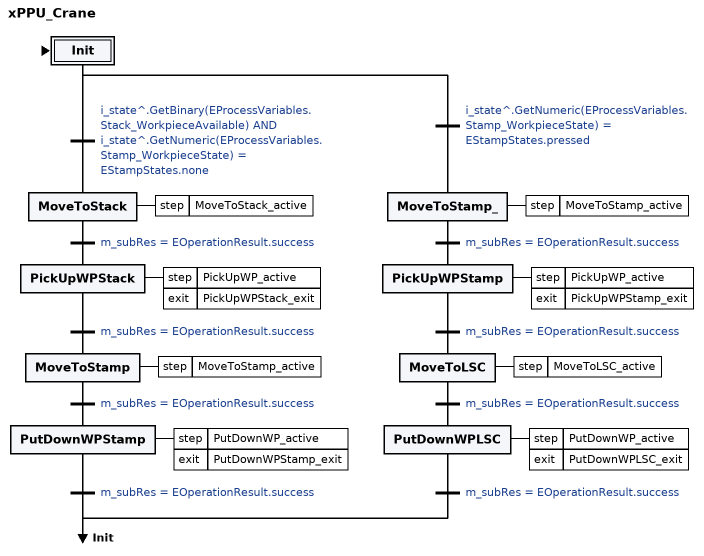
INITIAL_STEP Init:
END_STEP
TRANSITION FROM Init TO MoveToStack
    := i_state^.GetBinary(EProcessVariables.Stack_WorkpieceAvailable) AND i_state^.GetNumeric(EProcessVariables.Stamp_WorkpieceState) = EStampStates.none;
END_TRANSITION
STEP MoveToStack:
    MoveToStack_active(N);  // step action
END_STEP
TRANSITION FROM MoveToStack TO PickUpWPStack
    := m_subRes = EOperationResult.success;
END_TRANSITION
STEP PickUpWPStack:
    PickUpWP_active(N);  // step action
    PickUpWPStack_exit(P0);  // exit action
END_STEP
TRANSITION FROM PickUpWPStack TO MoveToStamp
    := m_subRes = EOperationResult.success;
END_TRANSITION
STEP MoveToStamp:
    MoveToStamp_active(N);  // step action
END_STEP
TRANSITION FROM MoveToStamp TO PutDownWPStamp
    := m_subRes = EOperationResult.success;
END_TRANSITION
STEP PutDownWPStamp:
    PutDownWP_active(N);  // step action
    PutDownWPStamp_exit(P0);  // exit action
END_STEP
TRANSITION FROM PutDownWPStamp TO Init
    := m_subRes = EOperationResult.success;
END_TRANSITION
TRANSITION FROM Init TO MoveToStamp_
    := i_state^.GetNumeric(EProcessVariables.Stamp_WorkpieceState) = EStampStates.pressed;
END_TRANSITION
STEP MoveToStamp_:
    MoveToStamp_active(N);  // step action
END_STEP
TRANSITION FROM MoveToStamp_ TO PickUpWPStamp
    := m_subRes = EOperationResult.success;
END_TRANSITION
STEP PickUpWPStamp:
    PickUpWP_active(N);  // step action
    PickUpWPStamp_exit(P0);  // exit action
END_STEP
TRANSITION FROM PickUpWPStamp TO MoveToLSC
    := m_subRes = EOperationResult.success;
END_TRANSITION
STEP MoveToLSC:
    MoveToLSC_active(N);  // step action
END_STEP
TRANSITION FROM MoveToLSC TO PutDownWPLSC
    := m_subRes = EOperationResult.success;
END_TRANSITION
STEP PutDownWPLSC:
    PutDownWP_active(N);  // step action
    PutDownWPLSC_exit(P0);  // exit action
END_STEP
TRANSITION FROM PutDownWPLSC TO Init
    := m_subRes = EOperationResult.success;
END_TRANSITION

ACTION MoveToLSC_active:
m_subRes := i_process^.Execute(
	EBehaviorType.control_primitive,
	EPrimitives.Crane_MoveToLSC,
	m_emptyParams);
END_ACTION

ACTION MoveToStack_active:
m_subRes := i_process^.Execute(
	EBehaviorType.control_primitive,
	EPrimitives.Crane_MoveToStack,
	m_emptyParams);
END_ACTION

ACTION MoveToStamp_active:
m_subRes := i_process^.Execute(
	EBehaviorType.control_primitive,
	EPrimitives.Crane_MoveToStamp,
	m_emptyParams);
END_ACTION

ACTION PickUpWP_active:
m_subRes := i_process^.Execute(
	EBehaviorType.control_primitive,
	EPrimitives.Crane_PickUpWP,
	m_emptyParams);
END_ACTION

ACTION PickUpWPStack_exit:
//i_state^.ShiftProduct(EProducts.stack_product, EProducts.crane_product);
END_ACTION

ACTION PickUpWPStamp_exit:
//i_state^.ShiftProduct(EProducts.stamp_product, EProducts.crane_product);
END_ACTION

ACTION PutDownWP_active:
m_subRes := i_process^.Execute(
	EBehaviorType.control_primitive,
	EPrimitives.Crane_PutDownWP,
	m_emptyParams);
END_ACTION

ACTION PutDownWPLSC_exit:
//i_state^.ShiftProduct(EProducts.crane_product, EProducts.LSC_product);
END_ACTION

ACTION PutDownWPStamp_exit:
//i_state^.ShiftProduct(EProducts.crane_product, EProducts.stamp_product);
END_ACTION

END_FUNCTION_BLOCK

// ---- POUs/01_SequenceControl/xPPU_Stamp.TcPOU
FUNCTION_BLOCK xPPU_Stamp
VAR_INPUT
	i_error: POINTER TO ErrorManager;
	i_process: POINTER TO ProcessManager;
	i_state: POINTER TO StateTracker;
END_VAR
VAR
	m_stampParams: ParameterSet;
	m_subRes: EOperationResult;
END_VAR

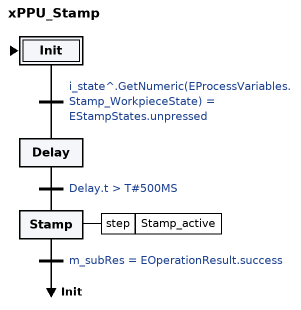
INITIAL_STEP Init:
END_STEP
TRANSITION FROM Init TO Delay
    := i_state^.GetNumeric(EProcessVariables.Stamp_WorkpieceState) = EStampStates.unpressed;
END_TRANSITION
STEP Delay:
END_STEP
TRANSITION FROM Delay TO Stamp
    := Delay.t > T#500MS;
END_TRANSITION
STEP Stamp:
    Stamp_active(N);  // step action
END_STEP
TRANSITION FROM Stamp TO Init
    := m_subRes = EOperationResult.success;
END_TRANSITION

ACTION Stamp_active:
m_stampParams.SetParam_Numeric('pressure_white', 4000);
m_stampParams.SetParam_Numeric('pressure_black', 4000);
m_stampParams.SetParam_Numeric('pressure_metal', 4000);

m_subRes := i_process^.Execute(
	EBehaviorType.control_primitive,
	EPrimitives.Stamp_StampWorkpiece,
	m_stampParams);
END_ACTION

END_FUNCTION_BLOCK

// ---- POUs/01_SequenceControl/xPPU_LSC.TcPOU
FUNCTION_BLOCK xPPU_LSC
VAR_INPUT
	i_error: POINTER TO ErrorManager;
	i_process: POINTER TO ProcessManager;
	i_state: POINTER TO StateTracker;
END_VAR
VAR
	m_conveyorParams: ParameterSet;
	m_subRes: EOperationResult;
END_VAR

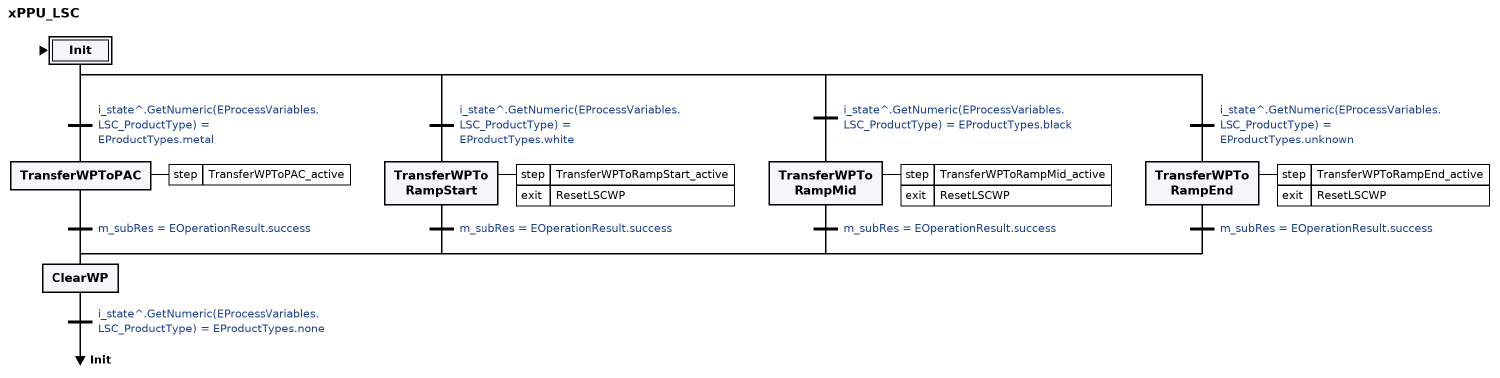
INITIAL_STEP Init:
END_STEP
TRANSITION FROM Init TO TransferWPToPAC
    := i_state^.GetNumeric(EProcessVariables.LSC_ProductType) = EProductTypes.metal;
END_TRANSITION
STEP TransferWPToPAC:
    TransferWPToPAC_active(N);  // step action
END_STEP
TRANSITION FROM TransferWPToPAC TO ClearWP
    := m_subRes = EOperationResult.success;
END_TRANSITION
TRANSITION FROM Init TO TransferWPToRampStart
    := i_state^.GetNumeric(EProcessVariables.LSC_ProductType) = EProductTypes.white;
END_TRANSITION
STEP TransferWPToRampStart:
    TransferWPToRampStart_active(N);  // step action
    ResetLSCWP(P0);  // exit action
END_STEP
TRANSITION FROM TransferWPToRampStart TO ClearWP
    := m_subRes = EOperationResult.success;
END_TRANSITION
TRANSITION FROM Init TO TransferWPToRampMid
    := i_state^.GetNumeric(EProcessVariables.LSC_ProductType) = EProductTypes.black;
END_TRANSITION
STEP TransferWPToRampMid:
    TransferWPToRampMid_active(N);  // step action
    ResetLSCWP(P0);  // exit action
END_STEP
TRANSITION FROM TransferWPToRampMid TO ClearWP
    := m_subRes = EOperationResult.success;
END_TRANSITION
TRANSITION FROM Init TO TransferWPToRampEnd
    := i_state^.GetNumeric(EProcessVariables.LSC_ProductType) = EProductTypes.unknown;
END_TRANSITION
STEP TransferWPToRampEnd:
    TransferWPToRampEnd_active(N);  // step action
    ResetLSCWP(P0);  // exit action
END_STEP
TRANSITION FROM TransferWPToRampEnd TO ClearWP
    := m_subRes = EOperationResult.success;
END_TRANSITION
STEP ClearWP:
END_STEP
TRANSITION FROM ClearWP TO Init
    := i_state^.GetNumeric(EProcessVariables.LSC_ProductType) = EProductTypes.none;
END_TRANSITION

ACTION ResetLSCWP:
i_state^.ShiftProduct(EProducts.LSC_product,0);
END_ACTION

ACTION TransferWPToPAC_active:
m_subRes := i_process^.Execute(
	EBehaviorType.control_primitive,
	EPrimitives.LSC_TransferWorkpieceTo_PAC,
	m_conveyorParams);
END_ACTION

ACTION TransferWPToRampEnd_active:
m_subRes := i_process^.Execute(
	EBehaviorType.control_primitive,
	EPrimitives.LSC_TransferWorkpieceTo_RampEnd,
	m_conveyorParams);
END_ACTION

ACTION TransferWPToRampMid_active:
m_subRes := i_process^.Execute(
	EBehaviorType.control_primitive,
	EPrimitives.LSC_TransferWorkpieceTo_RampMid,
	m_conveyorParams);
END_ACTION

ACTION TransferWPToRampStart_active:
m_subRes := i_process^.Execute(
	EBehaviorType.control_primitive,
	EPrimitives.LSC_TransferWorkpieceTo_RampStart,
	m_conveyorParams);
END_ACTION

END_FUNCTION_BLOCK

// ---- POUs/01_SequenceControl/xPPU_PAC.TcPOU
FUNCTION_BLOCK xPPU_PAC
VAR_INPUT
	i_error: POINTER TO ErrorManager;
	i_process: POINTER TO ProcessManager;
	i_state: POINTER TO StateTracker;
END_VAR
VAR
	m_emptyParams: ParameterSet;
	m_subRes: EOperationResult;
END_VAR

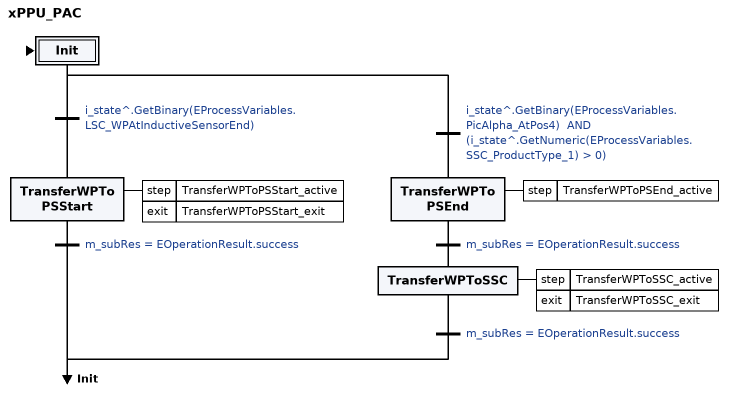
INITIAL_STEP Init:
END_STEP
TRANSITION FROM Init TO TransferWPToPSStart
    := i_state^.GetBinary(EProcessVariables.LSC_WPAtInductiveSensorEnd);
END_TRANSITION
STEP TransferWPToPSStart:
    TransferWPToPSStart_active(N);  // step action
    TransferWPToPSStart_exit(P0);  // exit action
END_STEP
TRANSITION FROM TransferWPToPSStart TO Init
    := m_subRes = EOperationResult.success;
END_TRANSITION
TRANSITION FROM Init TO TransferWPToPSEnd
    := i_state^.GetBinary(EProcessVariables.PicAlpha_AtPos4) AND (i_state^.GetNumeric(EProcessVariables.SSC_ProductType_1) > 0);
END_TRANSITION
STEP TransferWPToPSEnd:
    TransferWPToPSEnd_active(N);  // step action
END_STEP
TRANSITION FROM TransferWPToPSEnd TO TransferWPToSSC
    := m_subRes = EOperationResult.success;
END_TRANSITION
STEP TransferWPToSSC:
    TransferWPToSSC_active(N);  // step action
    TransferWPToSSC_exit(P0);  // exit action
END_STEP
TRANSITION FROM TransferWPToSSC TO Init
    := m_subRes = EOperationResult.success;
END_TRANSITION

ACTION TransferWPToPSEnd_active:
m_subRes := i_process^.Execute(
	EBehaviorType.control_primitive,
	EPrimitives.PAC_TransferWorkpieceTo_PSEnd,
	m_emptyParams);
END_ACTION

ACTION TransferWPToPSStart_active:
m_subRes := i_process^.Execute(
	EBehaviorType.control_primitive,
	EPrimitives.PAC_TransferWorkpieceTo_PSStart,
	m_emptyParams);
END_ACTION

ACTION TransferWPToPSStart_exit:
CASE LREAL_TO_INT(i_state^.GetNumeric(EProcessVariables.PAC_WPNumber)) OF
	1:	i_state^.ShiftProduct(EProducts.LSC_product, EProducts.PAC_product1);
	2:	i_state^.ShiftProduct(EProducts.LSC_product, EProducts.PAC_product2);
	3: 	i_state^.ShiftProduct(EProducts.LSC_product, EProducts.PAC_product3);
END_CASE
END_ACTION

ACTION TransferWPToSSC_active:
m_subRes := i_process^.Execute(
	EBehaviorType.control_primitive,
	EPrimitives.PAC_TransferWorkpieceTo_SSC,
	m_emptyParams);
END_ACTION

ACTION TransferWPToSSC_exit:
//shift products from PAC to SSC
i_state^.ShiftProduct(EProducts.PAC_product1, EProducts.SSC_product1);
i_state^.ShiftProduct(EProducts.PAC_product2, EProducts.SSC_product2);
END_ACTION

END_FUNCTION_BLOCK

// ---- POUs/01_SequenceControl/xPPU_PicAlpha.TcPOU
FUNCTION_BLOCK xPPU_PicAlpha
VAR_INPUT
	i_error: POINTER TO ErrorManager;
	i_process: POINTER TO ProcessManager;
	i_state: POINTER TO StateTracker;
END_VAR
VAR
	m_emptyParams: ParameterSet;
	m_subRes: EOperationResult;
END_VAR

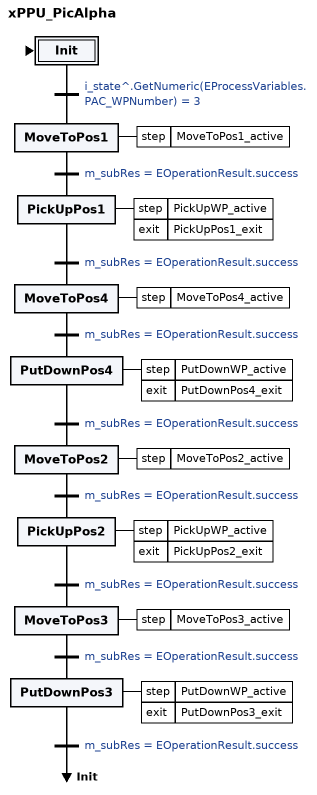
INITIAL_STEP Init:
END_STEP
TRANSITION FROM Init TO MoveToPos1
    := i_state^.GetNumeric(EProcessVariables.PAC_WPNumber) = 3;
END_TRANSITION
STEP MoveToPos1:
    MoveToPos1_active(N);  // step action
END_STEP
TRANSITION FROM MoveToPos1 TO PickUpPos1
    := m_subRes = EOperationResult.success;
END_TRANSITION
STEP PickUpPos1:
    PickUpWP_active(N);  // step action
    PickUpPos1_exit(P0);  // exit action
END_STEP
TRANSITION FROM PickUpPos1 TO MoveToPos4
    := m_subRes = EOperationResult.success;
END_TRANSITION
STEP MoveToPos4:
    MoveToPos4_active(N);  // step action
END_STEP
TRANSITION FROM MoveToPos4 TO PutDownPos4
    := m_subRes = EOperationResult.success;
END_TRANSITION
STEP PutDownPos4:
    PutDownWP_active(N);  // step action
    PutDownPos4_exit(P0);  // exit action
END_STEP
TRANSITION FROM PutDownPos4 TO MoveToPos2
    := m_subRes = EOperationResult.success;
END_TRANSITION
STEP MoveToPos2:
    MoveToPos2_active(N);  // step action
END_STEP
TRANSITION FROM MoveToPos2 TO PickUpPos2
    := m_subRes = EOperationResult.success;
END_TRANSITION
STEP PickUpPos2:
    PickUpWP_active(N);  // step action
    PickUpPos2_exit(P0);  // exit action
END_STEP
TRANSITION FROM PickUpPos2 TO MoveToPos3
    := m_subRes = EOperationResult.success;
END_TRANSITION
STEP MoveToPos3:
    MoveToPos3_active(N);  // step action
END_STEP
TRANSITION FROM MoveToPos3 TO PutDownPos3
    := m_subRes = EOperationResult.success;
END_TRANSITION
STEP PutDownPos3:
    PutDownWP_active(N);  // step action
    PutDownPos3_exit(P0);  // exit action
END_STEP
TRANSITION FROM PutDownPos3 TO Init
    := m_subRes = EOperationResult.success;
END_TRANSITION

ACTION MoveToPos1_active:
m_subRes := i_process^.Execute(
	EBehaviorType.control_primitive,
	EPrimitives.PicAlpha_MoveToPos1,
	m_emptyParams);
END_ACTION

ACTION MoveToPos2_active:
m_subRes := i_process^.Execute(
	EBehaviorType.control_primitive,
	EPrimitives.PicAlpha_MoveToPos2,
	m_emptyParams);
END_ACTION

ACTION MoveToPos3_active:
m_subRes := i_process^.Execute(
	EBehaviorType.control_primitive,
	EPrimitives.PicAlpha_MoveToPos3,
	m_emptyParams);
END_ACTION

ACTION MoveToPos4_active:
m_subRes := i_process^.Execute(
	EBehaviorType.control_primitive,
	EPrimitives.PicAlpha_MoveToPos4,
	m_emptyParams);
END_ACTION

ACTION PickUpPos1_exit:
i_state^.ShiftProduct(EProducts.PAC_product2, EProducts.PicAlpha_product);
i_state^.ShiftProduct(EProducts.PAC_product3, EProducts.PAC_product2);
END_ACTION

ACTION PickUpPos2_exit:
i_state^.ShiftProduct(EProducts.PAC_product2, EProducts.PicAlpha_product);
END_ACTION

ACTION PickUpWP_active:
m_subRes := i_process^.Execute(
	EBehaviorType.control_primitive,
	EPrimitives.PicAlpha_PickUpWP,
	m_emptyParams);
END_ACTION

ACTION PutDownPos3_exit:
i_state^.ShiftProduct(EProducts.PicAlpha_product, EProducts.PAC_product2);
END_ACTION

ACTION PutDownPos4_exit:
//shift product from PicAlpha to SSC
i_state^.ShiftProduct(EProducts.PicAlpha_product, EProducts.SSC_product1);
END_ACTION

ACTION PutDownWP_active:
m_subRes := i_process^.Execute(
	EBehaviorType.control_primitive,
	EPrimitives.PicAlpha_PutDownWp,
	m_emptyParams);
END_ACTION

END_FUNCTION_BLOCK

// ---- POUs/01_SequenceControl/xPPU_SSC.TcPOU
FUNCTION_BLOCK xPPU_SSC
VAR_INPUT
	i_error: POINTER TO ErrorManager;
	i_process: POINTER TO ProcessManager;
	i_state: POINTER TO StateTracker;
END_VAR
VAR
	m_emptyParams: ParameterSet;
	m_subRes: EOperationResult;
END_VAR

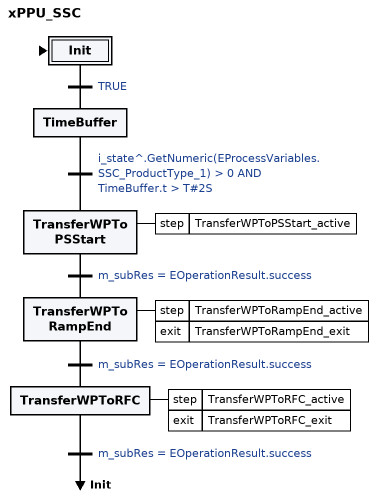
INITIAL_STEP Init:
END_STEP
TRANSITION FROM Init TO TimeBuffer
    := TRUE;
END_TRANSITION
STEP TimeBuffer:
END_STEP
TRANSITION FROM TimeBuffer TO TransferWPToPSStart
    := i_state^.GetNumeric(EProcessVariables.SSC_ProductType_1) > 0 AND TimeBuffer.t > T#2S;
END_TRANSITION
STEP TransferWPToPSStart:
    TransferWPToPSStart_active(N);  // step action
END_STEP
TRANSITION FROM TransferWPToPSStart TO TransferWPToRampEnd
    := m_subRes = EOperationResult.success;
END_TRANSITION
STEP TransferWPToRampEnd:
    TransferWPToRampEnd_active(N);  // step action
    TransferWPToRampEnd_exit(P0);  // exit action
END_STEP
TRANSITION FROM TransferWPToRampEnd TO TransferWPToRFC
    := m_subRes = EOperationResult.success;
END_TRANSITION
STEP TransferWPToRFC:
    TransferWPToRFC_active(N);  // step action
    TransferWPToRFC_exit(P0);  // exit action
END_STEP
TRANSITION FROM TransferWPToRFC TO Init
    := m_subRes = EOperationResult.success;
END_TRANSITION

ACTION TransferWPToPSStart_active:
m_subRes := i_process^.Execute(
	EBehaviorType.control_primitive,
	EPrimitives.SSC_TransferWorkpieceTo_PSStart,
	m_emptyParams);
END_ACTION

ACTION TransferWPToRampEnd_active:
m_subRes := i_process^.Execute(
	EBehaviorType.control_primitive,
	EPrimitives.SSC_TransferWorkpieceTo_RampEnd,
	m_emptyParams);
END_ACTION

ACTION TransferWPToRampEnd_exit:
i_state^.ShiftProduct(EProducts.SSC_product1,0);
END_ACTION

ACTION TransferWPToRFC_active:
m_subRes := i_process^.Execute(
	EBehaviorType.control_primitive,
	EPrimitives.SSC_TransferWorkpieceTo_RFC,
	m_emptyParams);
END_ACTION

ACTION TransferWPToRFC_exit:
i_state^.ShiftProduct(EProducts.SSC_product1, EProducts.RFC_product1);
i_state^.ShiftProduct(EProducts.SSC_product2, EProducts.RFC_product2);
END_ACTION

END_FUNCTION_BLOCK

// ---- POUs/01_SequenceControl/xPPU_RFC.TcPOU
FUNCTION_BLOCK xPPU_RFC
VAR_INPUT
	i_error: POINTER TO ErrorManager;
	i_process: POINTER TO ProcessManager;
	i_state: POINTER TO StateTracker;
END_VAR
VAR
	m_emptyParams: ParameterSet;
	m_subRes: EOperationResult;
END_VAR

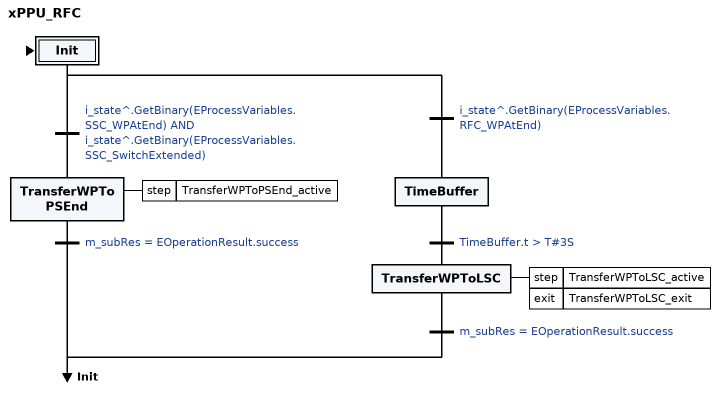
INITIAL_STEP Init:
END_STEP
TRANSITION FROM Init TO TransferWPToPSEnd
    := i_state^.GetBinary(EProcessVariables.SSC_WPAtEnd) AND i_state^.GetBinary(EProcessVariables.SSC_SwitchExtended);
END_TRANSITION
STEP TransferWPToPSEnd:
    TransferWPToPSEnd_active(N);  // step action
END_STEP
TRANSITION FROM TransferWPToPSEnd TO Init
    := m_subRes = EOperationResult.success;
END_TRANSITION
TRANSITION FROM Init TO TimeBuffer
    := i_state^.GetBinary(EProcessVariables.RFC_WPAtEnd);
END_TRANSITION
STEP TimeBuffer:
END_STEP
TRANSITION FROM TimeBuffer TO TransferWPToLSC
    := TimeBuffer.t > T#3S;
END_TRANSITION
STEP TransferWPToLSC:
    TransferWPToLSC_active(N);  // step action
    TransferWPToLSC_exit(P0);  // exit action
END_STEP
TRANSITION FROM TransferWPToLSC TO Init
    := m_subRes = EOperationResult.success;
END_TRANSITION

ACTION TransferWPToLSC_active:
m_subRes := i_process^.Execute(
	EBehaviorType.control_primitive,
	EPrimitives.RFC_TransferWorkpieceTo_LSC,
	m_emptyParams);
END_ACTION

ACTION TransferWPToLSC_exit:
i_state^.ShiftProduct(EProducts.RFC_product1, EProducts.LSC_product);
IF i_state^.GetBinary(EProcessVariables.RFC_WPAtEnd) THEN
	i_state^.ShiftProduct(EProducts.RFC_product2, EProducts.RFC_product1);
END_IF
END_ACTION

ACTION TransferWPToPSEnd_active:
m_subRes := i_process^.Execute(
	EBehaviorType.control_primitive,
	EPrimitives.RFC_TransferWorkpieceTo_PSEnd,
	m_emptyParams);
END_ACTION

END_FUNCTION_BLOCK

// ---- POUs/98_Utility/FC_InitAlarmTexts.TcPOU
FUNCTION FC_InitAlarmTexts : BOOL
VAR_INPUT
END_VAR
VAR
END_VAR

HMI_Texts.AlarmTexts[EAlarms.none] := 'unspecified';
HMI_Texts.AlarmTexts[EAlarms.initialized] := 'the component is not initialized yet';
HMI_Texts.AlarmTexts[EAlarms.did_execute] := 'the component executed';
HMI_Texts.AlarmTexts[EAlarms.stopped] := 'the system shut down';

HMI_Texts.AlarmTexts[ESpecialAlarmIds.recovery_request] := 'a recovery was requested';
HMI_Texts.AlarmTexts[ESpecialAlarmIds.definition_request] := 'a definition was requested';

END_FUNCTION
